FUNCTION_BLOCK FB_PCV
VAR_INPUT
END_VAR
VAR_OUTPUT
	bError : BOOL;
	nErrorId : ERRORID;
END_VAR
VAR
	bFill		: BOOL;
	tmrTimeout	: TON;
	bSensor		AT %I* : BOOL; 	//Verknüpfung mit Füllstandssensor
	bDigiOut 	AT %Q* : BOOL; 	//Verknüpfung muss mit Pumpe und StopVentil erfolgen
	bPneuValve	AT %Q* : BOOL;	//Verknüpfung mit Pneumatikventil (nur bei SolenoidPip)	
END_VAR

IF bSensor AND bFill THEN
	{IF defined(variable:cLiquidBottleNrPCV)}
	IF NOT aSensSysLiquidBottle[cLiquidBottleNrPCV] THEN //kein Systemwasser vorhanden
		bError := TRUE;
		nErrorId := E_ErrorIdCmd.ERRORID_LiquidBottleEmpty;
	END_IF
	{ELSE}
	IF NOT aSensSysLiquidBottle[1] THEN //kein Systemwasser vorhanden
		bError := TRUE;
		nErrorId := E_ErrorIdCmd.ERRORID_LiquidBottleEmpty;
	END_IF	
	{END_IF}

	IF NOT bError AND bFill THEN
		tmrTimeout(IN:= TRUE, PT:=T#1M);
		bDigiOut := TRUE;
	ELSE
		tmrTimeout(IN:= FALSE);
		bDigiOut := FALSE;	
	END_IF

	bFill := FALSE;
ELSE
	tmrTimeout(IN:= FALSE);
	bDigiOut := FALSE;	
	tmrTimeout(IN:= FALSE);
END_IF

IF tmrTimeout.Q THEN
	bError := TRUE;
	nErrorId := E_ErrorIdCmd.ERRORID_TimeOutFillPCV;
	bDigiOut := FALSE;
END_IF

METHOD M_Fill
VAR_INPUT
END_VAR
bFill := TRUE;
END_METHOD

METHOD M_Reset
VAR_INPUT
END_VAR
bError := FALSE;
END_METHOD

METHOD M_SwitchPneuValve
VAR_INPUT
	bOn : BOOL;
END_VAR
bPneuValve := bOn;
END_METHOD

PROPERTY P_bPneuValve : BOOL
GET
P_bPneuValve := bPneuValve;
END_GET
END_PROPERTY

END_FUNCTION_BLOCK

(* stored: Version 1.1.0.1
   POU FB_PCV: Id {74f59eec-ed0d-4676-9e92-6ecaab4452d6}, SpecialFunc None
   Method M_Fill: Id {54c8a2c6-8d9c-4e59-9062-1c031fc9e14c}
   Method M_Reset: Id {2484b465-5156-4f36-a325-b40c1a4d3f8f}
   Method M_SwitchPneuValve: Id {7996a399-e240-4868-b9ee-646a613b2001}
   Property P_bPneuValve: Id {446d3dd3-cd47-4d4e-abda-4ee30bc6917d}
   Get Get: Id {c7a289da-8557-48a2-bf86-f3bae11b3d3b} *)
